TYPE ST_ITC_TTA :
(**************************************************************************************
 * 	Application		:	BoxControl Framework
 *	Revision		:	$Revision: 404529 $
 *	Revision date	:	$Date: 2018-04-23 08:21:38 +0200 (Mo., 23 Apr 2018) $
 *	Last changed by	:	$Author: b7bolm $
 *	URL				:	$URL: http://almscdc.swisslog.com/repo/SWPD/Development/BoxControlFramework/20_Release/trunk/01_Software/BCF/BCF/JumpStart/20_Product/10_App/11_Com/10_Lib/10_Conv/11_ITC/01_DUTs/ST_ITC_TTA.TcDUT $
 *
 *	Purpose			:	ITC TTA Structure
 *
 * ------------------------------------------------------------------------------------
 *	Copyright Swisslog [IP AG], Switzerland. All rights reserved.
 * 
 * ------------------------------------------------------------------------------------
 *	
 * 	Revision History: 
 *
 * 	VERSION			DATE			INITIALS			DESCRIPTION
 *	0.1				01.01.2001		swl					Example
 *
 **************************************************************************************)
STRUCT
	Position				: STRING(Conveyor.POSITION_STRINGLENGTH); // 12 digit SIS location MM-GGG-EEEE-FF-Z 
	TU_DataIndex			: DINT; // 6 digit TU index
	MsgSequence				: INT; // 3 digit MSG sequence
	TU_ID					: STRING(Conveyor.TU_ID_STRINGLENGTH); // 18 digit TU ID 
	TU_Type					: INT; // 4 digit TU type 
	AssignmentID			: UDINT; // 8 digit assignment
	Length					: INT; // 4 digit dimension
	Width					: INT; // 4 digit dimension
	Height					: INT; // 4 digit dimension
	Weight					: DINT; // 8 digit weight
	Orientation				: STRING(Conveyor.ORIENTATION_STRINGLENGTH); // 3 digit orientation
	TU_Parameter 			: INT; // 4 digit parameter
	IO_Data					: INT; // 3 digit IO data 
	LowerLimit				: DINT; // 8 digit lower limit 
	UpperLimit				: DINT; // 8 digit upper limit 
	Sequence				: ULINT; // 19 digit global sequence identifier
	SubSequence				: DINT; // 9 digit position in the sequence
	SequenceSize			: DINT; // 9 digit number of TU's in the sequence
	GroupID					: ULINT; // 19 digit global group identifier 
	GroupSize				: DINT; // 9 digit number of TU's in the group ID
	DestinationSlot			: INT; // 3 digit logical sub destination of destination
	NumberOfDestinations	: INT; // 2 digit numner of destinations 
	Destination				: ARRAY [1..Conveyor.NUMBER_OF_DESTINATIONS] OF STRING(Conveyor.POSITION_STRINGLENGTH); // Array of 12 digit SIS destinations 
END_STRUCT
END_TYPE

(* stored: Version 1.1.0.1, ProductVersion 3.1.4022.12
   DUT ST_ITC_TTA: Id {1c7dc9b5-ec9b-4e69-87ca-4d5f90776f38} *)
